Staubli VAL3: initParams.pgx

public program initParams()
  local num l_nRetVal
begin
  l_nRetVal=sioCtrl(siTcpIpMotion,"timeout",2)
  if (l_nRetVal!=0)
    popUpMsg("Error while setting consumer timeout")
    //return ?
  endIf

  l_nRetVal=sioCtrl(siTcpIpFbk,"timeout",2)
  if (l_nRetVal!=0)
    popUpMsg("Error while setting producer timeout")
    //return ?
  endIf
end
